TYPE ST_SAFETY_FBTWOHAND:
STRUCT
	uStatus							: U_SAFETY_TWOHAND; 	(* Typ zalezny od bloku *)
	eState							: E_SAFETY_FBState;		(* Enum ze statusem bloku *)
	bGeneralError					: BOOL; 				(* Gdy wystapi chociaz jeden Error *)
END_STRUCT
END_TYPE

(* stored: Version 1.1.0.1, ProductVersion 3.1.4022.12
   DUT ST_SAFETY_FBTWOHAND: Id {761e870a-077d-49a9-9897-2389a0d0f0b2} *)
